FUNCTION_BLOCK Atuador_Pistao (* Template for a Basic Function Block Type *)
  (* Standard: 61499-2 *)
  (* Version 1.0, 2025-02-04, FESTO *)
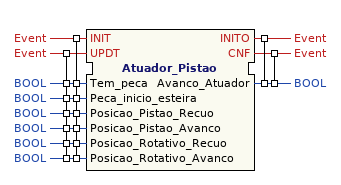
  EVENT_INPUT
    INIT WITH Tem_peca, Peca_inicio_esteira, Posicao_Pistao_Recuo, Posicao_Pistao_Avanco, Posicao_Rotativo_Recuo, Posicao_Rotativo_Avanco; (* Initialization Request *)
    UPDT WITH Tem_peca, Peca_inicio_esteira, Posicao_Pistao_Recuo, Posicao_Pistao_Avanco, Posicao_Rotativo_Recuo, Posicao_Rotativo_Avanco; (* Update *)
  END_EVENT
  EVENT_OUTPUT
    INITO WITH Avanco_Atuador; (* Initialization Confirm *)
    CNF WITH Avanco_Atuador; (* Execution Confirmation *)
  END_EVENT
  VAR_INPUT
    Tem_peca : BOOL; (* Verifica a presenca de peca no armazem. *)
    Peca_inicio_esteira : BOOL; (* Verifica a presenca de peca no início da esteira *)
    Posicao_Pistao_Recuo : BOOL;
    Posicao_Pistao_Avanco : BOOL;
    Posicao_Rotativo_Recuo : BOOL;
    Posicao_Rotativo_Avanco : BOOL;
  END_VAR
  VAR_OUTPUT
    Avanco_Atuador : BOOL; (* Output event qualifier *)
  END_VAR
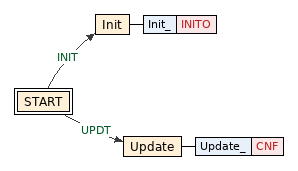
  EC_STATES
    START; (* Initial State *)
    Init : Init_ -> INITO;
    Update : Update_ -> CNF;
  END_STATES
  EC_TRANSITIONS
    START TO Init := INIT;
    START TO Update := UPDT;
  END_TRANSITIONS
  ALGORITHM Init_ IN ST:
	Avanco_Atuador:=FALSE;
  END_ALGORITHM
  ALGORITHM Update_ IN ST:
Avanco_Atuador:=FALSE;

IF Tem_Peca AND Posicao_Pistao_Recuo AND Posicao_Rotativo_Avanco THEN

Avanco_Atuador:=TRUE;

END_IF
  END_ALGORITHM
END_FUNCTION_BLOCK
